FUNCTION_BLOCK SLOT_SIMPLE_CIRCLE_SPLIT_DATA (* Splits data from iterator table for slot *)
  (* Standard: 61499-2 *)
  (* Version 1.0, 05-06-12, GASR, Universidade do Estado de Santa Catarina *)
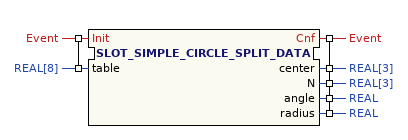
  EVENT_INPUT
    Init WITH table;
  END_EVENT
  EVENT_OUTPUT
    Cnf WITH center, N, angle, radius;
  END_EVENT
  VAR_INPUT
    table : ARRAY [0..7] OF REAL;
  END_VAR
  VAR_OUTPUT
    center : ARRAY [0..2] OF REAL;
    N : ARRAY [0..2] OF REAL;
    angle : REAL;
    radius : REAL;
  END_VAR
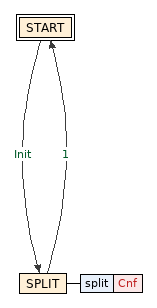
  EC_STATES
    START;
    SPLIT : split -> Cnf;
  END_STATES
  EC_TRANSITIONS
    START TO SPLIT := Init;
    SPLIT TO START := 1;
  END_TRANSITIONS
  ALGORITHM split IN Lua:
center[1] = table[1]
center[2] = table[2]
center[3] = table[3]
angle = table[4]
radius = table[5]
N[1] = table[6]
N[2] = table[7]
N[3] = table[8]
print( 'angle', angle, N[1], N[2], N[3] )
  END_ALGORITHM
END_FUNCTION_BLOCK
